FUNCTION_BLOCK ConveyorRingTokenCTL (* Basic Function Block Type *)
  (* Standard: 61499-2 *)
  (* Version 0.2, 2003-12-04, JHC, Rockwell Automation, Renamed for better indexing. *)
  (* Version 0.1, 2002-11-05, JHC, Rockwell Automation, Corrected missing ST element in Algorithm REQ. *)
  (* Version 0.0, 2000-05-30, JHC, Rockwell Automation *)
  (* Compiler header: package fb.rt.cs725; *)
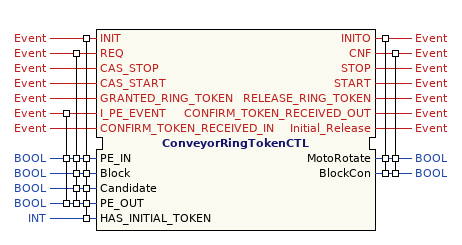
  EVENT_INPUT
    INIT WITH PE_IN, Block, Candidate, PE_OUT, HAS_INITIAL_TOKEN; (* Initialization Request *)
    REQ WITH Block, Candidate, PE_OUT, PE_IN; (* Normal Execution Request *)
    CAS_STOP;
    CAS_START;
    GRANTED_RING_TOKEN;
    I_PE_EVENT WITH PE_IN, PE_OUT;
    CONFIRM_TOKEN_RECEIVED_IN;
  END_EVENT
  EVENT_OUTPUT
    INITO WITH MotoRotate, BlockCon; (* Initialization Confirm *)
    CNF WITH MotoRotate, BlockCon; (* Execution Confirmation *)
    STOP;
    START;
    RELEASE_RING_TOKEN;
    CONFIRM_TOKEN_RECEIVED_OUT;
    Initial_Release;
  END_EVENT
  VAR_INPUT
    PE_IN : BOOL; (* Input event qualifier *)
    Block : BOOL;
    Candidate : BOOL;
    PE_OUT : BOOL;
    HAS_INITIAL_TOKEN : INT;
  END_VAR
  VAR_OUTPUT
    MotoRotate : BOOL; (* Output event qualifier *)
    BlockCon : BOOL;
  END_VAR
  VAR
    lastPE : BOOL := 1;
    lastBlock : BOOL := 0;
    hasInitialToken : BOOL;
  END_VAR
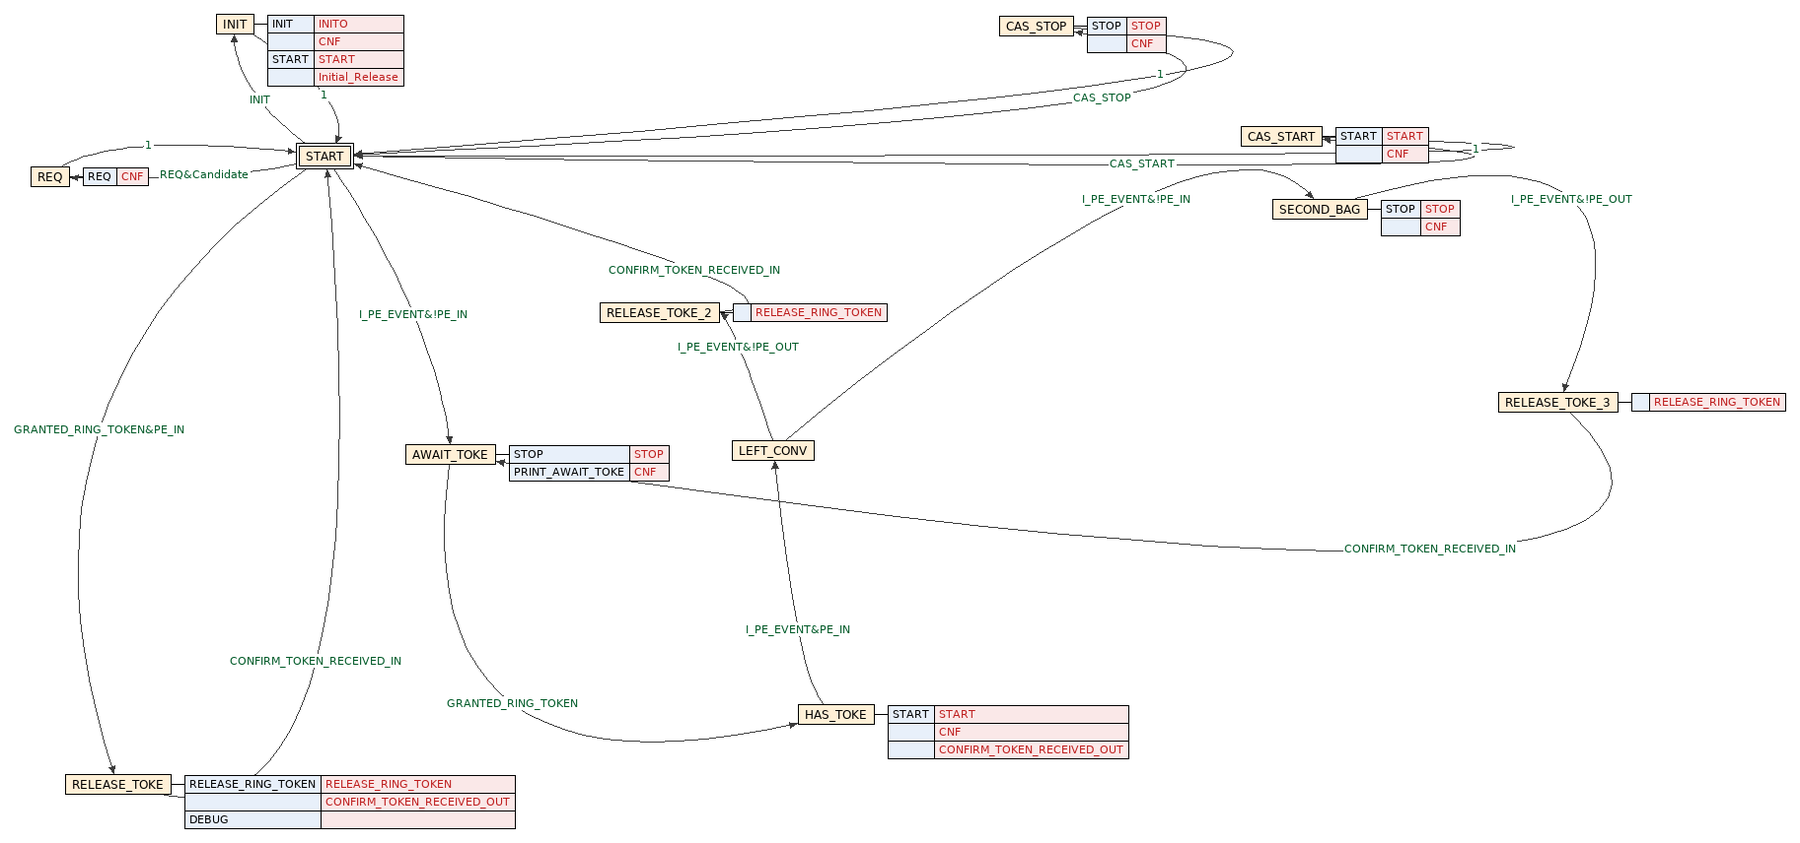
  EC_STATES
    START; (* Initial State *)
    INIT : INIT -> INITO, -> CNF, START -> START, -> Initial_Release; (* Initialization *)
    REQ : REQ -> CNF; (* Normal execution *)
    CAS_START : START -> START, -> CNF;
    CAS_STOP : STOP -> STOP, -> CNF;
    AWAIT_TOKE : STOP -> STOP, PRINT_AWAIT_TOKE -> CNF;
    RELEASE_TOKE : RELEASE_RING_TOKEN -> RELEASE_RING_TOKEN, -> CONFIRM_TOKEN_RECEIVED_OUT, DEBUG;
    LEFT_CONV;
    RELEASE_TOKE_2 : -> RELEASE_RING_TOKEN;
    HAS_TOKE : START -> START, -> CNF, -> CONFIRM_TOKEN_RECEIVED_OUT;
    SECOND_BAG : STOP -> STOP, -> CNF;
    RELEASE_TOKE_3 : -> RELEASE_RING_TOKEN;
  END_STATES
  EC_TRANSITIONS
    START TO INIT := INIT;
    START TO REQ := REQ&Candidate;
    REQ TO START := 1;
    START TO CAS_START := CAS_START;
    CAS_START TO START := 1;
    START TO CAS_STOP := CAS_STOP;
    CAS_STOP TO START := 1;
    START TO AWAIT_TOKE := I_PE_EVENT&!PE_IN;
    LEFT_CONV TO RELEASE_TOKE_2 := I_PE_EVENT&!PE_OUT;
    RELEASE_TOKE_2 TO START := CONFIRM_TOKEN_RECEIVED_IN;
    HAS_TOKE TO LEFT_CONV := I_PE_EVENT&PE_IN;
    AWAIT_TOKE TO HAS_TOKE := GRANTED_RING_TOKEN;
    LEFT_CONV TO SECOND_BAG := I_PE_EVENT&!PE_IN;
    SECOND_BAG TO RELEASE_TOKE_3 := I_PE_EVENT&!PE_OUT;
    RELEASE_TOKE_3 TO AWAIT_TOKE := CONFIRM_TOKEN_RECEIVED_IN;
    RELEASE_TOKE TO START := CONFIRM_TOKEN_RECEIVED_IN;
    START TO RELEASE_TOKE := GRANTED_RING_TOKEN&PE_IN;
    INIT TO START := 1;
  END_TRANSITIONS
  ALGORITHM INIT IN ST: (* Initialization algorithm *)
MotoRotate := TRUE;
Block := FALSE;

System.out.println(this + " " + MotoRotate);
System.out.println(MotoRotate);
System.out.println(this + "state of variable: " + HAS_INITIAL_TOKEN);
  END_ALGORITHM
  ALGORITHM REQ IN ST: (* Normally executed algorithm *)
//System.out.println(this +  " -> Candidate" + Candidate);
IF Candidate THEN
IF lastPE !:= PE_IN THEN
IF NOT PE_IN THEN
BlockCon:= TRUE;
System.out.println("BlockCon = true");
ELSE
BlockCon:=FALSE;
System.out.println("BlockCon = false");
END_IF
lastPE := PE_IN;
END_IF
IF lastBlock !:= Block THEN
IF Block THEN
STOP.serviceEvent(this);
MotoRotate := FALSE;
System.out.println("Cas Stop");
ELSE
START.serviceEvent(this);
MotoRotate := TRUE;
System.out.println("Cas Start");
END_IF
lastBlock := Block;
END_IF
END_IF
  END_ALGORITHM
  ALGORITHM START IN ST:
MotoRotate:=TRUE;
System.out.println(this + " Start " + MotoRotate);

System.out.println("Start " + MotoRotate);
  END_ALGORITHM
  ALGORITHM STOP IN ST:
MotoRotate := FALSE;
System.out.println(this + " Stop " + MotoRotate);

System.out.println("Stop " + MotoRotate);
  END_ALGORITHM
  ALGORITHM DEBUG IN ST:
System.out.println("release_toke state");
  END_ALGORITHM
  ALGORITHM RELEASE_RING_TOKEN IN ST:
System.out.println("Released the token!");
hasInitialToken := FALSE;
  END_ALGORITHM
  ALGORITHM RECEIVED_RING_TOKEN IN ST:
System.out.println("Received token!");
  END_ALGORITHM
  ALGORITHM PRINT_AWAIT_TOKE IN ST:
System.out.println("Awaiting token!");
  END_ALGORITHM
  ALGORITHM CHECK_IF_FIRST IN ST:

  END_ALGORITHM
END_FUNCTION_BLOCK
